FUNCTION_BLOCK FB_FireOffCommand IMPLEMENTS I_Command
VAR
	refFlameCannon : REFERENCE TO FB_FlameCannon;
END_VAR

METHOD Execute
IF (__ISVALIDREF(THIS^.refFlameCannon)) THEN
	THIS^.refFlameCannon.Off();
END_IF
END_METHOD

METHOD FB_init : BOOL
VAR_INPUT
	bInitRetains 	: BOOL; // if TRUE, the retain variables are initialized (warm start / cold start)
	bInCopyCode 	: BOOL;  // if TRUE, the instance afterwards gets moved into the copy code (online change)
	refFlameCannon 	: REFERENCE TO FB_FlameCannon;
END_VAR
IF (__ISVALIDREF(refFlameCannon)) THEN
	THIS^.refFlameCannon REF= refFlameCannon;
ELSE
	THIS^.refFlameCannon REF= 0;
END_IF
END_METHOD

END_FUNCTION_BLOCK

(* stored: Version 1.1.0.1, ProductVersion 3.1.4022.18
   POU FB_FireOffCommand: Id {714b9945-5f85-41e4-aa66-153e194c69f6}, SpecialFunc None
   Method Execute: Id {869ebaf8-c59a-472e-9c7f-510b734fe6d0}
   Method FB_init: Id {203782f2-4140-4af5-9c6a-bc1bfe74a5e7} *)
